SUBAPPLICATION Uebung_001 (* DigitalInput_I1 auf DigitalOutput_Q1 *)
  (* Standard: 61499-2 *)
  (* Version 1.0, 2023-10-23, franz *)
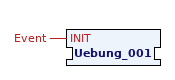
  EVENT_INPUT
    INIT;
  END_EVENT
END_SUBAPPLICATION
